(* IEC 61131-3 sources: DemoPumpStation/PumpStation/core/unit_manager, 6 files *)

(* ---- i_pump_units.st ---- *)
type
	unitHandle : ref_to PumpUnit;
end_type

interface IPumpUnits
	method init
		var_input
			collection : ref_to array[*] of PumpUnit;
			nominal_power : real;
		end_var
	end_method

	method getActiveCount : udint
	end_method

	method findNextAvailable : unitHandle
	end_method

	method findBypassUnit : unitHandle
	end_method

	method findUnit : unitHandle
	var_input id : udint; end_var
	end_method

	method getSize : udint
	end_method

	method getUnitRole : PumpRole
	var_input index : udint; end_var
	end_method

	method getUnitAvailable : bool
	var_input index : udint; end_var
	end_method

	method getUnitFaulted : bool
	var_input index : udint; end_var
	end_method

	method getUnitActive : bool
	var_input index : udint; end_var
	end_method

	method getCurrentPower : real
	var_input freq : real; end_var
	end_method

end_interface

(* ---- i_unit_manager.st ---- *)
type
	unitHandle : ref_to PumpUnit;
end_type

interface IUnitManager
	method init
		var_input
			collection : ref_to array[*] of PumpUnit;
			nominal_power : real;
		end_var
	end_method

	method getActiveCount : udint
	end_method

	method findNextAvailable : unitHandle
	end_method

	method findBypassUnit : unitHandle
	end_method

	method getSize : udint
	end_method

	method getUnitRole : PumpRole
	var_input index : udint; end_var
	end_method

	method getUnitAvailable : bool
	var_input index : udint; end_var
	end_method

	method getUnitFaulted : bool
	var_input index : udint; end_var
	end_method

	method getUnitActive : bool
	var_input index : udint; end_var
	end_method

	method getCurrentPower : real
	var_input freq : real; end_var
	end_method

end_interface

(* ---- i_controller_state.st ---- *)
interface IControllerState
    method isStarted : bool
    end_method

    method getRequestedPower : real
    end_method

    method getVfdUnitId : udint
    end_method
end_interface

(* ---- pump_unit.st ---- *)
class PumpUnit

var
    id : udint;
    role : PumpRole := PumpRole#stopped;
    available : bool := true;
    faulted : bool := false;
end_var

var private
	performance : real;
end_var

method public getPerformance : real
	var_input freq : real; end_var
	if role = PumpRole#stopped OR role = PumpRole#error then return;
	elseif role = PumpRole#onBypass then
		getPerformance := performance;
		return;
	else
		getPerformance := performance * (freq / 50.0);
	end_if
end_method

method public init
var_input
	unitId : udint;
	nominal : real;
end_var
	performance := nominal;
    id := unitId;
end_method

method public isActive : bool
    isActive := role <> PumpRole#stopped;
end_method

end_class

(* ---- pump_units_manager.st ---- *)
class UnitManager implements IPumpUnits
	var private
		units : ref_to array[*] of PumpUnit;
		start, end : udint;
		size : udint;
	end_var

	method private isValid : bool
		if units = NULL then return; end_if
		if size = 0 then return; end_if
		isValid := true;
	end_method

	method public init
		var_input
			collection : ref_to array[*] of PumpUnit;
			nominal_power : real;
		end_var
		var i : udint; end_var

		if collection = NULL then return; end_if
		start := lower_bound(collection, 1);
		end := upper_bound(collection, 1);
		size := 1 + end - start;
		units := collection;

		for i := start to end do
        	units^[i].init(i - start + 1, nominal_power);
    	end_for

	end_method

	method public getActiveCount : udint
	var i : udint; cnt : udint; end_var
	    for i := start to end do
	        if units^[i].isActive() then
	            cnt := cnt + 1;
	        end_if
	    end_for
	    getActiveCount := cnt;
	end_method

	method findUnit : unitHandle
	var_input id : udint; end_var
	var i : udint; end_var
	    for i := start to end do
	        if units^[i].id = id then
	            findUnit := ref(units^[i]);
	            return;
	        end_if
	    end_for
	end_method

	method public findNextAvailable : unitHandle
	var i : udint; end_var
		if not this.isValid() then return; end_if

	    for i := start to end do
	        if units^[i].available and not units^[i].faulted and not units^[i].isActive() then
	        	findNextAvailable := ref(units^[i]);
	            return;
	        end_if
	    end_for
	end_method

	method public findBypassUnit : unitHandle
	var i : udint; end_var
		if not this.isValid() then return; end_if
	    for i := start to end do
	        if units^[i].role = PumpRole#onBypass then
	        	findBypassUnit := ref(units^[i]);
	            return;
	        end_if
	    end_for
	end_method

	method getSize : udint
		getSize := size;
	end_method

	method public getUnitRole : PumpRole
	var_input i : udint; end_var
		getUnitRole := PumpRole#error;
		if not this.isValid() then return; end_if

	    for i := start to end do
	        if units^[i].id = i then
	        	getUnitRole := units^[i].role;
	            return;
	        end_if
	    end_for
	end_method

	method public getUnitAvailable : bool
	var_input i : udint; end_var

		if not this.isValid() then return; end_if

	    for i := start to end do
	        if units^[i].id = i then
	        	getUnitAvailable := units^[i].available;
	            return;
	        end_if
	    end_for

	end_method

	method public getUnitFaulted : bool
	var_input i : udint; end_var

	    getUnitFaulted := true;
		if not this.isValid() then return; end_if

	    for i := start to end do
	        if units^[i].id = i then
	        	getUnitFaulted := units^[i].faulted;
	            return;
	        end_if
	    end_for

	end_method

	method public getUnitActive : bool
	var_input i : udint; end_var

		if not this.isValid() then return; end_if

	    for i := start to end do
	        if units^[i].id = i then
	        	getUnitActive := units^[i].isActive();
	            return;
	        end_if
	    end_for
	end_method

	method getCurrentPower : real
	var_input freq : real; end_var
	var i : udint; end_var
		if not this.isValid() then return; end_if
	    for i := start to end do
		    getCurrentPower := getCurrentPower + units^[i].getPerformance(freq);
	    end_for
	end_method

end_class

(* ---- unit_manager.st ---- *)
class UnitManager implements IUnitManager
	var private
		units : ref_to array[*] of PumpUnit;
		start, end : udint;
		size : udint;
	end_var

	method private isValid : bool
		if units = NULL then return; end_if
		if size = 0 then return; end_if
		isValid := true;
	end_method

	method public init
		var_input
			collection : ref_to array[*] of PumpUnit;
			nominal_power : real;
		end_var
		var i : udint; end_var

		if collection = NULL then return; end_if
		start := lower_bound(collection, 1);
		end := upper_bound(collection, 1);
		size := 1 + end - start;
		units := collection;

		for i := start to end do
        	units^[i].init(i - start + 1, nominal_power);
    	end_for

	end_method

	method public getActiveCount : udint
	var i : udint; cnt : udint; end_var
	    for i := start to end do
	        if units^[i].isActive() then
	            cnt := cnt + 1;
	        end_if
	    end_for
	    getActiveCount := cnt;
	end_method

	method public findNextAvailable : unitHandle
	var i : udint; end_var
		if not this.isValid() then return; end_if

	    for i := start to end do
	        if units^[i].available and not units^[i].faulted and not units^[i].isActive() then
	        	findNextAvailable := ref(units^[i]);
	            return;
	        end_if
	    end_for
	end_method

	method public findBypassUnit : unitHandle
	var i : udint; end_var
		if not this.isValid() then return; end_if
	    for i := start to end do
	        if units^[i].role = PumpRole#onBypass then
	        	findBypassUnit := ref(units^[i]);
	            return;
	        end_if
	    end_for
	end_method

	method getSize : udint
		getSize := size;
	end_method

	method public getUnitRole : PumpRole
	var_input i : udint; end_var
		getUnitRole := PumpRole#error;
		if not this.isValid() then return; end_if

	    for i := start to end do
	        if units^[i].id = i then
	        	getUnitRole := units^[i].role;
	            return;
	        end_if
	    end_for
	end_method

	method public getUnitAvailable : bool
	var_input i : udint; end_var

		if not this.isValid() then return; end_if

	    for i := start to end do
	        if units^[i].id = i then
	        	getUnitAvailable := units^[i].available;
	            return;
	        end_if
	    end_for

	end_method

	method public getUnitFaulted : bool
	var_input i : udint; end_var

	    getUnitFaulted := true;
		if not this.isValid() then return; end_if

	    for i := start to end do
	        if units^[i].id = i then
	        	getUnitFaulted := units^[i].faulted;
	            return;
	        end_if
	    end_for

	end_method

	method public getUnitActive : bool
	var_input i : udint; end_var

		if not this.isValid() then return; end_if

	    for i := start to end do
	        if units^[i].id = i then
	        	getUnitActive := units^[i].isActive();
	            return;
	        end_if
	    end_for
	end_method

	method getCurrentPower : real
	var_input freq : real; end_var
	var i : udint; end_var
		if not this.isValid() then return; end_if
	    for i := start to end do
		    getCurrentPower := getCurrentPower + units^[i].getPerformance(freq);
	    end_for
	end_method

end_class
